FUNCTION_BLOCK FB_ControlLoop_MainPumpPressure

VAR
	{attribute 'OPC.UA.DA' := '0'}
	fbMainPump:  		I_PumpVSD;
	
	eSMState: 					(INIT, WAIT_TRIG, WAIT, CALCULATE) := INIT;
	
	eState_MaxHeadofOpenValve:  	(RECIRC, L1, L2, L3, L4, L5, L6, L7, L8, L9 , L10, L11, L12, L13, L14, L15, L16, L17, L18, L19, L20) := L1;
	bEnabled: BOOL := TRUE;
	bError: BOOL := FALSE;
	
	{attribute 'OPC.UA.DA' := '0'}
	fbTON_LoopTime: TON := (PT := T#1S);
	
END_VAR

VAR_IN_OUT
	setPointPressure: UINT := 0; // kPa 
	
END_VAR

fbTON_LoopTime();

CASE eSmstate OF
	
	INIT:

		eSMState := WAIT_TRIG;

	WAIT_TRIG:
	
		eSMState := WAIT;
	
	WAIT:
		IF fbTON_LoopTime.Q THEN
			fbTON_LoopTime(IN := FALSE);
			eSMState := CALCULATE;
		END_IF

	CALCULATE:
	
		IF eState_MaxHeadofOpenValve = RECIRC THEN
			setPointPressure := 200;
		ELSE
			CASE eState_MaxHeadofOpenValve OF
				L1: 
					setPointPressure := 270;
				L2: 
					setPointPressure := 340;
				L3: 
					setPointPressure := 410;
				L4: 
					setPointPressure := 480;
				L5: 
					setPointPressure := 550;
				L6: 
					setPointPressure := 620;
				L7: 
					setPointPressure := 690;
				L8: 
					setPointPressure := 760;
				L9: 
					setPointPressure := 830;
				L10: 
					setPointPressure := 900;
				L11: 
					setPointPressure := 970;
				L12: 
					setPointPressure := 1040;
				L13: 
					setPointPressure := 1100;
				L14: 
					setPointPressure := 1180;
				L15: 
					setPointPressure := 1250;
				L16: 
					setPointPressure := 1320;
				L17: 
					setPointPressure := 1390;
				L18: 
					setPointPressure := 1460;
				L19: 
					setPointPressure := 1530;
				L20: 
					setPointPressure := 1600;
				
			END_CASE
		END_IF
						

		eSMState := WAIT_TRIG;
END_CASE

METHOD FB_init : BOOL
VAR_INPUT
	bInitRetains : BOOL; // if TRUE, the retain variables are initialized (warm start / cold start)
	bInCopyCode : BOOL;  // if TRUE, the instance afterwards gets moved into the copy code (online change)
	
	MainPump:  		I_PumpVSD;
	
END_VAR
fbMainPump := MainPump;
END_METHOD

METHOD setCurrentLevel : BOOL
VAR_INPUT
	HighestLevel: UINT;
END_VAR

eState_MaxHeadofOpenValve := HighestLevel;
END_METHOD

END_FUNCTION_BLOCK

(* stored: Version 1.1.0.1, ProductVersion 3.1.4024.12
   POU FB_ControlLoop_MainPumpPressure: Id {4831c561-1bc0-41da-9721-e76b34f47b04}, SpecialFunc None
   Method FB_init: Id {d9a5effe-f158-4c3c-b566-c35dfefbe8e4}
   Method setCurrentLevel: Id {07362376-a9ff-451c-b800-ed7f3c8f70d4} *)
